// TIA Portal V17 export
// export: Created 2022-06-16T09:21:07.7045551Z, ExportSetting WithDefaults, DisplayName Totally Integrated Automation Portal, DisplayVersion V17, DisplayName TIA Portal Openness, DisplayVersion V17, DisplayName TIA Portal Version Control Interface, DisplayVersion V17, DisplayName STEP 7 Professional, DisplayVersion V17, DisplayName STEP 7 Safety, DisplayVersion V17, DisplayName WinCC Advanced, DisplayVersion V17
TYPE "typeScaleParam"
// stored: IsFailsafeCompliant false
   STRUCT
      axisNum : Int;
      "a" : Real;
      "b" : Real;
   END_STRUCT;
END_TYPE
